// TIA Portal V20 export
TYPE "LER_typeServoTorqueCalCommands"
// stored: Access Published
   STRUCT
      Reset : Bool;
      Save : Bool;
   END_STRUCT;
END_TYPE
